Universal Robots PolyScope program: align for floor straight.urp

Program align for floor straight (installation=default directory=/programs createdIn=5.21.3 lastSavedIn=5.21.3 robotSerialNumber=20246801938)
Calibrated DH parameters: a=[-0.000071, -0.790281, -0.600694, 0.000061, -0.000039, 0]; d=[0.236272, 604.465945, 132.116513, -736.382239, 0.159268, 0.154005]; alpha=[1.570254, -0.000567, 0.000559, 1.571709, -1.56999, 0]; deltaTheta=[0, -0.409357, 7.293326, -0.600784, -0.000001, -0.000001]
InitVariablesNode
Robot Program (runOnlyOnce=true)
  SuppressedNode
    Folder dummypoints
      MoveJ speed 60 deg/s, acceleration 80 deg/s^2 (useActiveTCP=true optimoveEnabled=false optiMoveSpeed=0.3 optiMoveAcceleration=0.09) feature=Base
        Waypoint oldhome: TCP in base x=397.354 y=356.263 z=319.809 mm, rx=2.3163 ry=2.0576 rz=0.0741 rad; joints [-198.308, -118.162, 133.452, -12.561, -11.517, -6.326] deg; TCP offset x=-9.5 y=-328 z=105.73 mm, rx=1.2092 ry=-1.2092 rz=1.2092 rad
        Waypoint demo: TCP in base x=-1245.427 y=-117.911 z=443.767 mm, rx=0.1153 ry=3.1146 rz=0.2657 rad; joints [0.095, -71.189, 81.089, -9.527, 94.427, -9.693] deg
        Waypoint Waypoint_1: TCP in base x=-262.599 y=-117.911 z=443.767 mm, rx=0.1153 ry=3.1146 rz=0.2657 rad; joints [5.497, -142.032, 129.309, 13.11, 99.793, -9.621] deg
  MoveJ speed 60 deg/s, acceleration 80 deg/s^2 (useActiveTCP=true optimoveEnabled=false optiMoveSpeed=0.3 optiMoveAcceleration=0.09) feature=Base
    Waypoint Waypoint_2: TCP in base x=397.354 y=356.263 z=319.809 mm, rx=2.3163 ry=2.0576 rz=0.0741 rad; joints [-198.308, -118.162, 133.452, -12.561, -11.517, -6.326] deg
    SuppressedNode
      Waypoint Waypoint_3: TCP in base x=-262.599 y=-117.911 z=443.767 mm, rx=0.1153 ry=3.1146 rz=0.2657 rad; joints [5.497, -142.032, 129.309, 13.11, 99.793, -9.621] deg
    Waypoint Waypoint_4: TCP in base x=-367.892 y=771.856 z=513.017 mm, rx=-2.0385 ry=0.4357 rz=2.0275 rad; joints [-102.301, -102.141, 125.99, -111.196, -90.364, -80.654] deg
    SuppressedNode
      Waypoint Waypoint_5: TCP in base x=-1242.22 y=568.091 z=-33.064 mm, rx=-2.1743 ry=0.2124 rz=2.1517 rad; joints [-41.317, -49.183, 112.752, -151.502, -88.354, -32.672] deg
    SuppressedNode
      Waypoint Waypoint_6: TCP in base x=-1225.108 y=565.114 z=-32.931 mm, rx=-2.1792 ry=0.203 rz=2.157 rad; joints [-41.957, -49.673, 114.09, -152.333, -88.377, 326.165] deg
    SuppressedNode
      Waypoint Waypoint_8: TCP in base x=-19.355 y=402.131 z=623.797 mm, rx=0.9216 ry=1.4113 rz=-2.2931 rad; joints [-129.203, -95.837, 121.075, -82.918, -50.734, 159.545] deg
    SuppressedNode
      Waypoint Waypoint_7: TCP in base x=-386.029 y=627.538 z=519.706 mm, rx=2.1582 ry=0.0261 rz=-2.169 rad; joints [-102.301, -102.141, 125.989, -111.196, -90.363, 253.708] deg
